//{attribute 'qualified_only'}
VAR_GLOBAL
	fbFEEDER: FB_FEEDER;
	fbSEPARATE1: FB_SEPARATE;
	fbSEPARATE2: FB_SEPARATE;
	LIFT1:FB_Axis;
	XY1:FB_Axis;
	LIFT2:FB_Axis;
	XY2:FB_Axis;
	PIST1: FB_PISTON;
	PIST2: FB_PISTON;
	PIST_FEEDER1: FB_PISTON;
	PIST_FEEDER2: FB_PISTON;
	PIST_FEEDER3: FB_PISTON;
	PIST_SEPARATE1_1: FB_PISTON;
	PIST_SEPARATE1_2: FB_PISTON;
	PIST_SEPARATE1_3: FB_PISTON;
	PIST_SEPARATE1_4: FB_PISTON;
	PIST_SEPARATE1_5: FB_PISTON;
	PIST_SEPARATE1_6: FB_PISTON;
	PIST_SEPARATE2_1: FB_PISTON;
	PIST_SEPARATE2_2: FB_PISTON;
	PIST_SEPARATE2_3: FB_PISTON;
	PIST_SEPARATE2_4: FB_PISTON;
	PIST_SEPARATE2_5: FB_PISTON;
	PIST_SEPARATE2_6: FB_PISTON;
	ACTION1:FB_ACTION;
	ACTION2:FB_ACTION;
END_VAR

(* stored: Version 1.1.0.1, ProductVersion 3.1.4024.12
   GVL GVL_MAIN: Id {7384caef-394f-40b5-a173-7cc02d269eff} *)
